# EPICS autosave request: ipApp/Db/InstekGPP_settings.req
# FILE... InstekGPP_settings.req
$(P)$(R)CH1_Vmeas.SCAN
$(P)$(R)CH1_Vmeas.DESC
$(P)$(R)CH1_Vset
$(P)$(R)CH1_V_TweakVal
$(P)$(R)CH1_Vlimit_Set
$(P)$(R)CH1_Iset
$(P)$(R)CH1_I_TweakVal
$(P)$(R)CH1_Ilimit_Set
$(P)$(R)CH2_Vmeas.DESC
$(P)$(R)CH2_Vset
$(P)$(R)CH2_V_TweakVal
$(P)$(R)CH2_Vlimit_Set
$(P)$(R)CH2_Iset
$(P)$(R)CH2_I_TweakVal
$(P)$(R)CH2_Ilimit_Set
